TYPE U_OdriveSetInputPosBytes :
UNION
    stSetInputPos : ST_OdriveSetInputPos;
    aBytes : ARRAY[0..7] OF BYTE;
END_UNION
END_TYPE

(* stored: Version 1.1.0.1
   DUT U_OdriveSetInputPosBytes: Id {099f976b-8a44-49c4-905b-1db7719026b0} *)
